// TIA Portal V16 export
// export: Created 2023-03-29T11:03:47.3458891Z, ExportSetting WithDefaults, DisplayName Totally Integrated Automation Portal, DisplayVersion V16 Update 6, DisplayName TIA Portal Version Control Interface, DisplayVersion V16 Update 2, DisplayName TIA Portal Openness, DisplayVersion V16 Update 6, DisplayName STEP 7 Professional, DisplayVersion V16 Update 6, DisplayName STEP 7 Safety, DisplayVersion V16, DisplayName WinCC Advanced, DisplayVersion V16 Update 6
TYPE "typeMbClient"
// stored: IsFailsafeCompliant false
   STRUCT
      req : Bool;   // Activates the requested transmission if TRUE
      disconnect : Bool;   // Initiates a disconnect operation
      mode : USInt;   // Specifies the type of request: read, write or diagnostic
      mbDataAddr : UDInt := 40066;   // Specifies the starting address of the data to be accessed in the Modbus client
      connect { S7_SetPoint := 'True'} : TCON_IP_v4;   // Reference to the connection parameters
   END_STRUCT;
   // connect.InterfaceId := 64;
   // connect.ID := 1;
   // connect.ActiveEstablished := true;
   // connect.RemoteAddress.ADDR[1] := 192;
   // connect.RemoteAddress.ADDR[2] := 168;
   // connect.RemoteAddress.ADDR[3] := 0;
   // connect.RemotePort := 502;
END_TYPE
